{attribute addProperty BoxType "EL1258-0000-0016"}
{attribute addProperty Id "Input_buffer_resetBIT10.1251Input_order_counterUSINT8117"}
{attribute addProperty CRC "760561105"}
{attribute addProperty SizeInBites "137"}
{attribute addProperty SizeInBytes "17.125"}
{warning 'Size of this structure is not a multiple of 8 bits!!!'}
TYPE Ctrl_2D553DD1 :
STRUCT
	{attribute addProperty Name "Input_buffer_reset"}
	Input_buffer_reset : BIT;
	{attribute 'hide'}
	reserve_1_BOOL_0 : BOOL;
	{attribute 'hide'}
	reserve_1_BOOL_1 : BOOL;
	{attribute 'hide'}
	reserve_1_BOOL_2 : BOOL;
	{attribute 'hide'}
	reserve_1_BOOL_3 : BOOL;
	{attribute 'hide'}
	reserve_1_BOOL_4 : BOOL;
	{attribute 'hide'}
	reserve_1_BOOL_5 : BOOL;
	{attribute 'hide'}
	reserve_1_BOOL_6 : BOOL;
	{attribute 'hide'}
	reserve_1_BOOL_7 : BOOL;
	{attribute 'hide'}
	reserve_1_BOOL_8 : BOOL;
	{attribute 'hide'}
	reserve_1_BOOL_9 : BOOL;
	{attribute 'hide'}
	reserve_1_BOOL_10 : BOOL;
	{attribute 'hide'}
	reserve_1_BOOL_11 : BOOL;
	{attribute 'hide'}
	reserve_1_BOOL_12 : BOOL;
	{attribute 'hide'}
	reserve_1_BOOL_13 : BOOL;
	{attribute 'hide'}
	reserve_1_BOOL_14 : BOOL;
	{attribute addProperty Name "Input_order_counter"}
	Input_order_counter : USINT;
	{attribute 'hide'}
	reserve_2 : BYTE;
END_STRUCT
END_TYPE

(* stored: Version 1.2.0.0, ProductVersion 3.1.4024.9
   DUT Ctrl_2D553DD1: Id {75b83bbb-3331-4dc9-b571-3a7c09f0d369} *)
